(* IEC 61131-3 sources: moqui-plc/simatic-ax/src-manual/framework/src/main/org/moqui/device, 2 files *)

(* ---- ParseRecipeDInt.st ---- *)
USING System.Strings;

FUNCTION ParseRecipeDInt : DINT
	VAR_INPUT
		value : STRING;
	END_VAR
	VAR_TEMP
		position : INT;
		startPosition : INT := INT#1;
		charText : STRING[1];
		sign : DINT := DINT#1;
		digit : DINT;
		valueLength : INT;
	END_VAR

	valueLength := LengthOf(value);
	IF valueLength <= INT#0 THEN
		RETURN;
	END_IF;

	charText := Substring(value, INT#1, INT#1);
	IF charText = '-' THEN
		sign := -DINT#1;
		startPosition := INT#2;
	ELSIF charText = '+' THEN
		startPosition := INT#2;
	END_IF;

	FOR position := startPosition TO valueLength DO
		charText := Substring(value, position, INT#1);
		CASE charText OF
			'0' : digit := DINT#0;
			'1' : digit := DINT#1;
			'2' : digit := DINT#2;
			'3' : digit := DINT#3;
			'4' : digit := DINT#4;
			'5' : digit := DINT#5;
			'6' : digit := DINT#6;
			'7' : digit := DINT#7;
			'8' : digit := DINT#8;
			'9' : digit := DINT#9;
		ELSE
			EXIT;
		END_CASE;
		ParseRecipeDInt := (ParseRecipeDInt * DINT#10) + digit;
	END_FOR;

	ParseRecipeDInt := ParseRecipeDInt * sign;
END_FUNCTION

(* ---- ParseRecipeReal.st ---- *)
USING System.Strings;

FUNCTION ParseRecipeReal : REAL
	VAR_INPUT
		value : STRING;
	END_VAR
	VAR_TEMP
		position : INT;
		startPosition : INT := INT#1;
		charText : STRING[1];
		sign : REAL := REAL#1.0;
		digit : REAL;
		decimalSeen : BOOL;
		fractionScale : REAL := REAL#1.0;
		valueLength : INT;
	END_VAR

	valueLength := LengthOf(value);
	IF valueLength <= INT#0 THEN
		RETURN;
	END_IF;

	charText := Substring(value, INT#1, INT#1);
	IF charText = '-' THEN
		sign := REAL#-1.0;
		startPosition := INT#2;
	ELSIF charText = '+' THEN
		startPosition := INT#2;
	END_IF;

	FOR position := startPosition TO valueLength DO
		charText := Substring(value, position, INT#1);
		IF charText = '.' THEN
			decimalSeen := TRUE;
		ELSE
			CASE charText OF
				'0' : digit := REAL#0.0;
				'1' : digit := REAL#1.0;
				'2' : digit := REAL#2.0;
				'3' : digit := REAL#3.0;
				'4' : digit := REAL#4.0;
				'5' : digit := REAL#5.0;
				'6' : digit := REAL#6.0;
				'7' : digit := REAL#7.0;
				'8' : digit := REAL#8.0;
				'9' : digit := REAL#9.0;
			ELSE
				EXIT;
			END_CASE;

			IF NOT decimalSeen THEN
				ParseRecipeReal := (ParseRecipeReal * REAL#10.0) + digit;
			ELSE
				fractionScale := fractionScale * REAL#10.0;
				ParseRecipeReal := ParseRecipeReal + (digit / fractionScale);
			END_IF;
		END_IF;
	END_FOR;

	ParseRecipeReal := ParseRecipeReal * sign;
END_FUNCTION
